Universal Robots PolyScope program: Step Corner Under L.urp

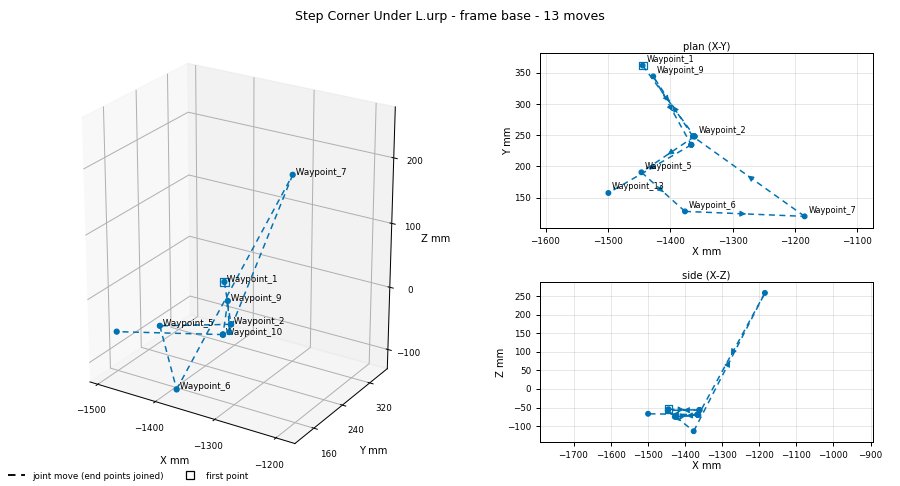
[picture p0: tool path of Step Corner Under L.urp in frame base, 13 of 13 moves have a stored position in this frame; points joined in program order, loops and branches not executed]
Program Step Corner Under L (installation=default directory=/programs createdIn=5.21.3 lastSavedIn=5.21.3 robotSerialNumber=20246801938)
Calibrated DH parameters: a=[-0.000071, -0.790281, -0.600694, 0.000061, -0.000039, 0]; d=[0.236272, 604.465945, 132.116513, -736.382239, 0.159268, 0.154005]; alpha=[1.570254, -0.000567, 0.000559, 1.571709, -1.56999, 0]; deltaTheta=[0, -0.409357, 7.293326, -0.600784, -0.000001, -0.000001]
InitVariablesNode
Robot Program (runOnlyOnce=false)
  Folder dummy points
    MoveJ speed 60 deg/s, acceleration 80 deg/s^2 (useActiveTCP=true optimoveEnabled=false optiMoveSpeed=0.3 optiMoveAcceleration=0.09) feature=Base
      Waypoint Waypoint_1: TCP in base x=-1444.215 y=361.78 z=-54.625 mm, rx=0.0014 ry=0.0235 rz=-2.509 rad; joints [-31.627, -5.956, 54.684, -47.848, 22.19, -181.767] deg; TCP offset x=-9.5 y=-328 z=105.73 mm, rx=1.2092 ry=-1.2092 rz=1.2092 rad
      Waypoint Waypoint_2: TCP in base x=-1360.959 y=248.194 z=-56.963 mm, rx=0.0014 ry=0.0235 rz=-2.509 rad; joints [-29.114, -11.124, 70.476, -58.547, 24.705, -181.685] deg
      Waypoint Waypoint_3: TCP in base x=-1360.959 y=248.194 z=-56.963 mm, rx=-0.0054 ry=0.0265 rz=-3.0281 rad; joints [-24.957, -13.827, 80.465, -66.855, 58.598, -180.908] deg
      Waypoint Waypoint_4: TCP in base x=-1360.959 y=248.194 z=-56.963 mm, rx=0.0148 ry=-0.0161 rz=2.1655 rad; joints [-11.656, -11.684, 73.347, -63.083, 134.303, -181.338] deg
      Waypoint Waypoint_5: TCP in base x=-1446.158 y=190.559 z=-57.572 mm, rx=0.0148 ry=-0.0161 rz=2.1655 rad; joints [-8.338, -8.416, 62.959, -56.049, 137.618, -181.456] deg
    'first one got very tight at the end of pivot rotation'
    'try 2'
    MoveJ speed 60 deg/s, acceleration 80 deg/s^2 (useActiveTCP=true optimoveEnabled=false optiMoveSpeed=0.3 optiMoveAcceleration=0.09) feature=Base
      Waypoint Waypoint_6: TCP in base x=-1376.345 y=127.862 z=-113.809 mm, rx=0.0016 ry=0.0206 rz=2.8022 rad; joints [-12.569, -10.644, 79.226, -68.552, 96.921, -179.181] deg
    'try 3'
    MoveJ speed 60 deg/s, acceleration 80 deg/s^2 (useActiveTCP=true optimoveEnabled=false optiMoveSpeed=0.3 optiMoveAcceleration=0.09) feature=Base
      Waypoint Waypoint_7: TCP in base x=-1184.505 y=119.919 z=258.583 mm, rx=-0.0165 ry=0.0559 rz=2.5896 rad; joints [-10.765, -17.591, 98.739, 100.27, -110.852, -357.508] deg
    MoveJ speed 60 deg/s, acceleration 80 deg/s^2 (useActiveTCP=true optimoveEnabled=false optiMoveSpeed=0.3 optiMoveAcceleration=0.09) feature=Base
      Waypoint Waypoint_8: TCP in base x=-1363.711 y=248.048 z=-70.154 mm, rx=-0.0362 ry=0.0515 rz=2.4999 rad; joints [-14.347, 7.149, 61.129, 114.102, -112.38, -357.575] deg
    MoveJ speed 60 deg/s, acceleration 80 deg/s^2 (useActiveTCP=true optimoveEnabled=false optiMoveSpeed=0.3 optiMoveAcceleration=0.09) feature=Base
      'this is the correct section of points'
      Waypoint Waypoint_9: TCP in base x=-1427.208 y=344.39 z=-74.96 mm, rx=0.0662 ry=-0.047 rz=-2.6322 rad; joints [-30.748, 12.35, 43.663, 128.657, -30.19, -1.48] deg
      Waypoint Waypoint_10: TCP in base x=-1366.187 y=234.655 z=-69.225 mm, rx=0.0662 ry=-0.047 rz=-2.6322 rad; joints [-27.63, 7.951, 57.667, 118.66, -33.302, -1.026] deg
      Waypoint Waypoint_11: TCP in base x=-1366.187 y=234.655 z=-69.225 mm, rx=-0.0864 ry=0.0277 rz=3.0352 rad; joints [-21.358, 5.615, 66.496, 111.398, -74.707, -0.173] deg
      Waypoint Waypoint_12: TCP in base x=-1366.187 y=234.655 z=-69.225 mm, rx=-0.0513 ry=0.0508 rz=2.097 rad; joints [-9.299, 8.891, 53.248, 122.982, -140.418, 4.749] deg
      Waypoint Waypoint_13: TCP in base x=-1499.166 y=157.371 z=-66.883 mm, rx=-0.0513 ry=0.0508 rz=2.097 rad; joints [-5.098, 16.63, 29.832, 139.174, -144.594, 5.408] deg
